(*These are parameters that are used to initiate axis movements
They are commands that are commonly used commands*)
TYPE ST_AxisControl :
STRUCT
    //Actions from controls system
    bExecute: BOOL; //Rising edge to execute some motion FB's
    bReset: BOOL; //Reset axis from Error state
    bStop: BOOL;
    bHalt: BOOL;
    bEnable: BOOL; //Enable axis drive
    bJogFwd: BOOL;
    bJogBwd: BOOL;
    bInterlockFwd: BOOL := FALSE; //Bit for interlocking motors in the positive direction
    bInterlockBwd: BOOL := FALSE; //Bit for interlocking motors in the negative direction
    eCommand: E_MotionFunctions;
    fVelocity: LREAL; //Velocity must be specified
    fJogVelocity: LREAL; //Jogging velocity
    fAcceleration: LREAL; //Not all FBs use, 0 is NC default
    fDeceleration: LREAL;
    fPosition: LREAL; //The position to move to for an absolute move and the amount to move in a relative move
	fRelativePosition: LREAL; //Position for relative moves
	fSetPosition : LREAL;
	bReinitialiseNcParameters : BOOL;
	
	bOverrideLimits : BOOL;
	
	bAutoEnableDisable : BOOL;
	
	bOverrideReadyToMove : BOOL;
	bExtReadyToMove : BOOL;
	tMoveFinishedDelay : TIME := T#1S;
END_STRUCT
END_TYPE

(* stored: Version 1.1.0.1, ProductVersion 3.1.4026.18
   DUT ST_AxisControl: Id {c02b2c99-be98-4acd-b0cb-dc10c1ff77f2} *)
